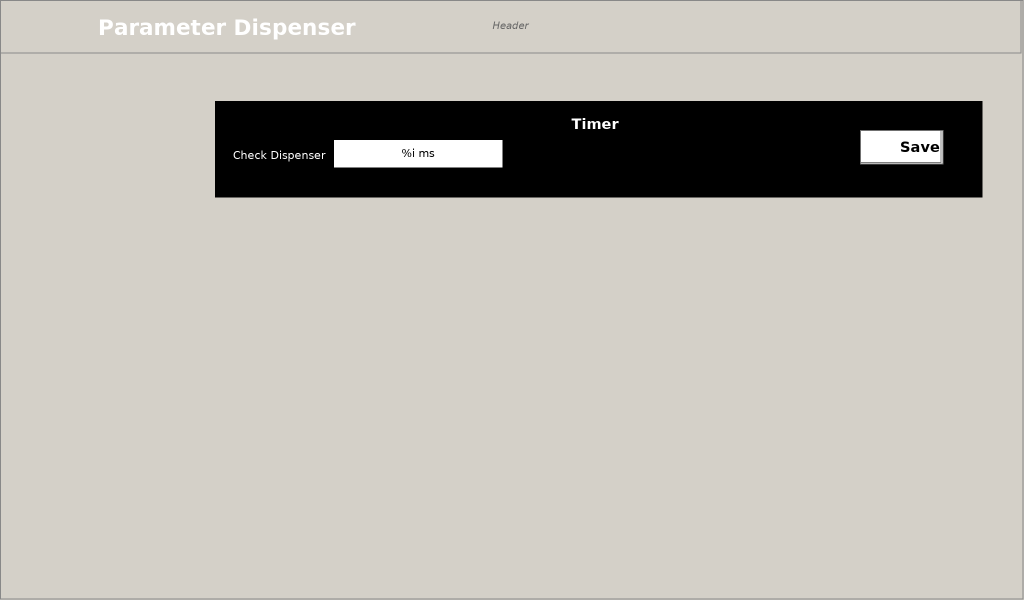
VISUALIZATION MDispenser  // 1024x600
    Frame (0,-2 1021x55)
        shows Header()
    Label (95,15 250x25), "Parameter Dispenser"
    RoundedRectangle (215,101 767x96)
    Label (243,104 704x40), "Timer"
    Label (230,138 103x35), "Check Dispenser"
    RoundedRectangle (333,139 170x29), "%i ms", text variable: HMI_GVL.Tmr_Dispenser
        OnMouseClick: write the text variable via Default
    Button (860,130 83x34), "Save", image: VisuSymbols.Symbols.Save
        tap InputOutput_GVL.TestMode[100]
END_VISUALIZATION

(* stored: Version 1.1.0.1, ProductVersion 3.1.4024.12
   Visu MDispenser: Id {369d4be4-2517-4ca5-850a-4510ea4b21c5} *)
